FUNCTION_BLOCK T_MockCommandTask IMPLEMENTS I_Task
VAR_INPUT
  _Busy, _Done, _Error, _Timeout : BOOL;
  _Result : LREAL;
END_VAR

METHOD Abort
END_METHOD

PROPERTY Available : BOOL
GET
END_GET
END_PROPERTY

PROPERTY Busy : BOOL
GET
Busy := _Busy;
END_GET
END_PROPERTY

METHOD CyclicLogic
END_METHOD

PROPERTY Done : BOOL
GET
Done := _Done;
END_GET
END_PROPERTY

PROPERTY Error : BOOL
GET
Error := _Error;
END_GET
END_PROPERTY

PROPERTY ErrorId : STRING
GET
END_GET
END_PROPERTY

METHOD Execute : BOOL
END_METHOD

METHOD Free
END_METHOD

PROPERTY Timeout : BOOL
GET
Timeout := _Timeout;
END_GET
END_PROPERTY

END_FUNCTION_BLOCK

(* stored: Version 1.1.0.1
   POU T_MockCommandTask: Id {e907346f-a42d-4c5a-a427-677e1fe4bdc3}, SpecialFunc None
   Method Abort: Id {3f2e672f-7fae-4734-84b2-99c8c0a8c445}
   Property Available: Id {06c58e6d-7319-46c6-a21d-04f63d55a421}
   Get Get: Id {5a1b141e-5ed8-4fe0-80fd-e6e0f88f2fec}
   Property Busy: Id {a42db8f4-a18d-48dd-a3dc-7bbdf1fac5ff}
   Get Get: Id {4e463914-63c3-4dec-9ab6-46f5d980f5b2}
   Method CyclicLogic: Id {8bf70dea-9862-426e-a39c-e83a4f2f93bc}
   Property Done: Id {59a1686f-35c1-4cdd-9ea5-aca27344b807}
   Get Get: Id {2af91fec-7ea1-4e0d-b7e3-61a04acaff85}
   Property Error: Id {7b14124c-44bb-4753-88bd-e895b6fe0d37}
   Get Get: Id {119fbfd4-7c5d-43fd-9d44-c90d4aceb44d}
   Property ErrorId: Id {6d290924-c9e0-4d88-9b1c-dbbce1b395e4}
   Get Get: Id {752053d6-3ff5-4217-9ddf-06f8914ac37f}
   Method Execute: Id {6347ddee-4222-4b08-9bfc-d8153a635e3c}
   Method Free: Id {c40a38ea-0515-429d-b1dd-948c4f8ea998}
   Property Timeout: Id {814a249d-148a-4ce7-9559-39d7d40a3770}
   Get Get: Id {8e0a93b1-371c-4ffb-b3aa-c000e1055f6c} *)
